{attribute 'qualified_only'}
VAR_GLOBAL
stHMIVaribles		: ST_CraneHMIData;
END_VAR

(* stored: Version 1.1.0.1, ProductVersion 3.1.4024.12
   GVL G_HMI: Id {72720ed5-c85c-48c4-b589-a11e5f3f0d01} *)
